INTERFACE I_CH_Object EXTENDS __SYSTEM.IQueryInterface

METHOD Initialize : HRESULT
END_METHOD

{attribute 'monitoring':='call'}
PROPERTY LUID : STRING //Locally unique identifier
GET
END_GET
END_PROPERTY

{attribute 'monitoring':='call'}
PROPERTY OID : OTCID //Object ID
GET
END_GET
END_PROPERTY

METHOD Update : HRESULT
VAR_INPUT
END_VAR
END_METHOD

END_INTERFACE

(* stored: Version 1.1.0.1, ProductVersion 3.1.4024.12
   Itf I_CH_Object: Id {b12f0d54-c62f-4bd7-8469-766bc19f5ddf}
   Method Initialize: Id {257a79bb-a0a4-4f1e-bf59-fa138996cb7c}
   Property LUID: Id {0a8cefee-5069-4827-8218-849224d67929}
   Get Get: Id {00c396d8-9d3e-4897-bdf9-5c6a0bb194fe}
   Property OID: Id {b43449ff-a0c9-4fe7-9dd9-24b5b0a7d8e6}
   Get Get: Id {2f46fd06-50e6-48ce-97a4-ffb4d8af9760}
   Method Update: Id {bb2c794e-2d3a-4108-8f6b-7a86da6d2da1} *)
